{attribute 'qualified_only'}
VAR_GLOBAL
	StateManager 	: StateManager;
END_VAR

(* stored: Version 1.1.0.1, ProductVersion 3.1.4022.11
   GVL Comp02: Id {22c97eee-6fba-4ca1-84b5-97f90bc5048d} *)
